// TIA Portal V16 export
// export: Created 2021-10-20T13:42:00.78736Z, ExportSetting WithDefaults, DisplayName Totally Integrated Automation Portal, DisplayVersion V16, DisplayName TIA Portal Version Control Interface, DisplayVersion V16, DisplayName TIA Portal Openness, DisplayVersion V16, DisplayName TIA Portal Teamcenter Gateway, DisplayVersion V16, DisplayName SINAMICS Startdrive Advanced, DisplayVersion V16, DisplayName SINAMICS Startdrive G130, G150, S120, S150, SINAMICS MV, S210, DisplayVersion V16, DisplayName SINAMICS Startdrive G110M, G120, G120C, G120D, G120P, DisplayVersion V16, DisplayName STEP 7 Professional, DisplayVersion V16, DisplayName STEP 7 Safety, DisplayVersion V16, DisplayName WinCC Advanced, DisplayVersion V16
ORGANIZATION_BLOCK "Main"   // OB1, LAD, ProgramCycle
TITLE = "Main Program Sweep (Cycle)"
{ S7_Optimized_Access := 'TRUE' }
VERSION : 0.1
// stored: AutoNumber true, IsIECCheckEnabled false, SetENOAutomatically false
   VAR_INPUT
      Initial_Call : Bool;   // Initial call of this OB
      Remanence : Bool;   // =True, if remanent data are available
   END_VAR
BEGIN

REGION Network 1: Call HART routine
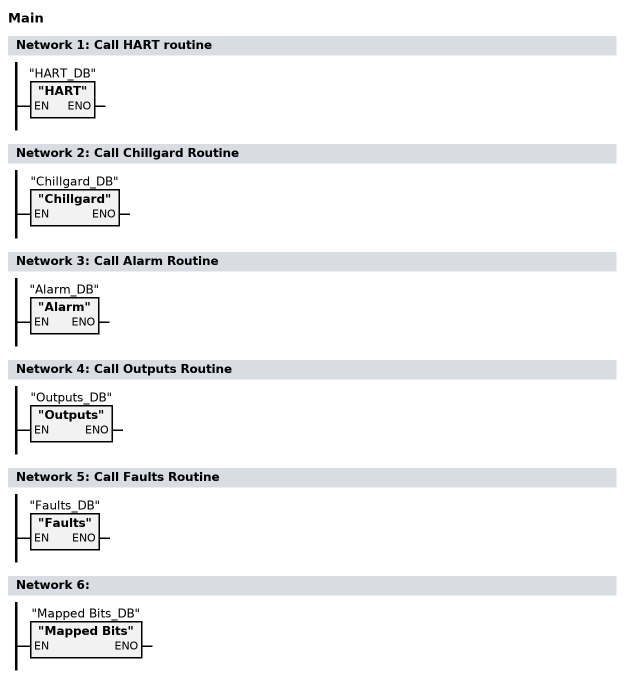
   RUNG wire#powerrail
      "HART_DB"()
   END_RUNG
   // the same network as SCL:
   "HART_DB"();   // "HART"
END_REGION

REGION Network 2: Call Chillgard Routine
   RUNG wire#powerrail
      "Chillgard_DB"()
   END_RUNG
   // the same network as SCL:
   "Chillgard_DB"();   // "Chillgard"
END_REGION

REGION Network 3: Call Alarm Routine
   RUNG wire#powerrail
      "Alarm_DB"()
   END_RUNG
   // the same network as SCL:
   "Alarm_DB"();   // "Alarm"
END_REGION

REGION Network 4: Call Outputs Routine
   RUNG wire#powerrail
      "Outputs_DB"()
   END_RUNG
   // the same network as SCL:
   "Outputs_DB"();   // "Outputs"
END_REGION

REGION Network 5: Call Faults Routine
   RUNG wire#powerrail
      "Faults_DB"()
   END_RUNG
   // the same network as SCL:
   "Faults_DB"();   // "Faults"
END_REGION

REGION Network 6
   RUNG wire#powerrail
      "Mapped Bits_DB"()
   END_RUNG
   // the same network as SCL:
   "Mapped Bits_DB"();   // "Mapped Bits"
END_REGION
END_ORGANIZATION_BLOCK
